FUNCTION_BLOCK RemoveAllMoverFromGroup  IMPLEMENTS I_Task
VAR
	RemoveAllFromGrp			: MC_UngroupAllAxes;
	_caGroup			: I_CollisionGroup;
	_Done 				: BOOL;
	_Error				: BOOL;
	_ErrorID			: UDINT;
END_VAR

{analysis -2}

METHOD Abort : BOOL
RemoveAllFromGrp.Execute := FALSE;
Abort := true;
END_METHOD

PROPERTY Busy : BOOL
GET
Busy := RemoveAllFromGrp.Busy;
END_GET
END_PROPERTY

METHOD Cycle : HRESULT
VAR_INPUT
END_VAR
IF _caGroup = 0 THEN
	Cycle := -1;
	RETURN;
END_IF

_Done := RemoveAllFromGrp.Done OR _Done;
_Error := RemoveAllFromGrp.Error OR _Error;
IF RemoveAllFromGrp.ErrorId <> 0 THEN
	_ErrorId := RemoveAllFromGrp.ErrorId;
END_IF
RemoveAllFromGrp(AxesGroup := _caGroup.GroupRef);
RemoveAllFromGrp.Execute := FALSE;
END_METHOD

PROPERTY Done : BOOL
GET
Done := _Done;
END_GET
END_PROPERTY

PROPERTY Error : BOOL
GET
Error := _Error;
END_GET
END_PROPERTY

PROPERTY MyCollisionGroup : I_CollisionGroup
GET
MyCollisionGroup := _caGroup;
END_GET
SET
IF MyCollisionGroup <> 0 THEN
	_caGroup := MyCollisionGroup;
END_IF
END_SET
END_PROPERTY

METHOD RemoveAllMover : HRESULT
IF RemoveAllFromGrp.Execute THEN
	RemoveAllMover := -1;
	RETURN;
END_IF
	
IF _caGroup = 0 THEN
	RemoveAllMover := -2;
	RETURN;
END_IF

RemoveAllFromGrp.Execute := TRUE;
END_METHOD

END_FUNCTION_BLOCK

(* stored: Version 1.1.0.1
   POU RemoveAllMoverFromGroup: Id {1511d483-7397-4cd0-a6db-08dd652e8cbb}, SpecialFunc None
   Method Abort: Id {e7050a73-9e5f-49ae-8033-79483a14dcd8}
   Property Busy: Id {0d92caac-9bc0-454c-a618-8bcbd6fddbf0}
   Get Get: Id {b2be66ef-24ca-4f17-b275-22f37a693e1a}
   Method Cycle: Id {c68e4170-0a2c-460f-9ca9-a0eca48c8c15}
   Property Done: Id {975b270f-4493-4b56-b51c-510ba823888a}
   Get Get: Id {95b9fdb8-73f9-4ddb-bfc3-1e9d09e71602}
   Property Error: Id {db24f627-0029-4f0f-a1df-743d439176a7}
   Get Get: Id {5d6c2566-9991-444d-a2dc-e184008251a9}
   Property MyCollisionGroup: Id {648a0ebd-d48b-4f7d-8cf0-533de95e54f9}
   Get Get: Id {047a9927-cc59-4451-88c4-bc2ec66e5e78}
   Set Set: Id {bc0a67ea-d15d-45ca-af76-84a2bf2313ea}
   Method RemoveAllMover: Id {0b41790b-140c-4897-91fc-096c85c5f45b} *)
